Fanuc KAREL source: V_CSAPI_SETVALUE.kl

PROGRAM T
%NOLOCKGROUP
VAR
 v0 : STRING[40]
 v1 : STRING[40]
 v2 : REAL
 v3 : INTEGER
BEGIN
 V_CSAPI_SETVALUE(v0, v1, v2, v3)
END T
